TYPE ST_Point :
STRUCT
x: int;
y: int;
END_STRUCT
END_TYPE

(* stored: Version 1.1.0.1
   DUT ST_Point: Id {p} *)
